// TIA Portal project "3_Queue_of_Items" (V19)

(* hardware
DEVICE "S7-1500/ET200MP station_1"  S7-1500 station
   slot 0: "Rail_0"  Rack  6ES7 590-1***0-0AA0
   slot 1: "PLC_1"  CPU 1513-1 PN  6ES7 513-1AL02-0AB0  V2.9
      slot 3: "CPU display_1"  6ES7591-1AA00-0AA0
      slot 32768: "PROFINET interface_1"  X1
         slot 32769: "Port_1"  X1 P1
         slot 32770: "Port_2"  X1 P2
      slot 34817: "Virtual CP interface port_1"  Virtual CP interface port  Virtual CP interface port
*)

// ===== PLC "PLC_1"  CPU 1513-1 PN =====

VAR_GLOBAL   // PLC tag table "Default tag table"
   "NGE_I0.3_Buffer" AT %M0.0 : Bool;
   "PE_Buffer_Conveyor" AT %M0.1 : Bool;
   "NE_Buffer_Conveyor" AT %M0.2 : Bool;
   "NE_Entry" AT %M0.3 : Bool;
   "NE_Exit" AT %M0.4 : Bool;
END_VAR

VAR_GLOBAL   // PLC tag table "Tag table from XML_1"
   "Start Button 1" AT %I0.0 : Bool;
   "Stop Button 1" AT %I0.1 : Bool;
   "Item Ready" AT %I0.2 : Bool;
   "At Entry" AT %I0.3 : Bool;
   "At Exit" AT %I0.4 : Bool;
   "Start Button 1 (Light)" AT %Q0.0 : Bool;
   "Stop Button 1 (Light)" AT %Q0.1 : Bool;
   "Entry conveyor" AT %Q0.2 : Bool;
   "Buffer conveyor" AT %Q0.3 : Bool;
   "Digital Display 1" AT %QD30 : DInt;
END_VAR

// folder: System blocks/Program resources

DATA_BLOCK "IEC_Counter_0_DB"   // DB1
{ S7_Optimized_Access := 'TRUE' }
AUTHOR : Simatic
FAMILY : IEC
NAME : CNTR
VERSION : 1.0
// stored: InstanceOfName IEC_COUNTER
"IEC_COUNTER"
BEGIN
END_DATA_BLOCK

DATA_BLOCK "IEC_Counter_0_DB_1"   // DB2
{ S7_Optimized_Access := 'TRUE' }
AUTHOR : Simatic
FAMILY : IEC
NAME : CNTR
VERSION : 1.0
// stored: InstanceOfName IEC_COUNTER
"IEC_COUNTER"
BEGIN
END_DATA_BLOCK

// folder: (top level)

ORGANIZATION_BLOCK "Main"   // OB1, LAD, ProgramCycle
TITLE = "Main Program Sweep (Cycle)"
{ S7_Optimized_Access := 'TRUE' }
VERSION : 0.1
   VAR_INPUT
      Initial_Call : Bool;   // Initial call of this OB
      Remanence : Bool;   // =True, if remanent data are available
   END_VAR
   VAR_TEMP   // added for the SCL form of the ladder/FBD networks
      _w1 : Bool;
      _w2 : Bool;
   END_VAR
BEGIN

REGION Network 1: Initial condition
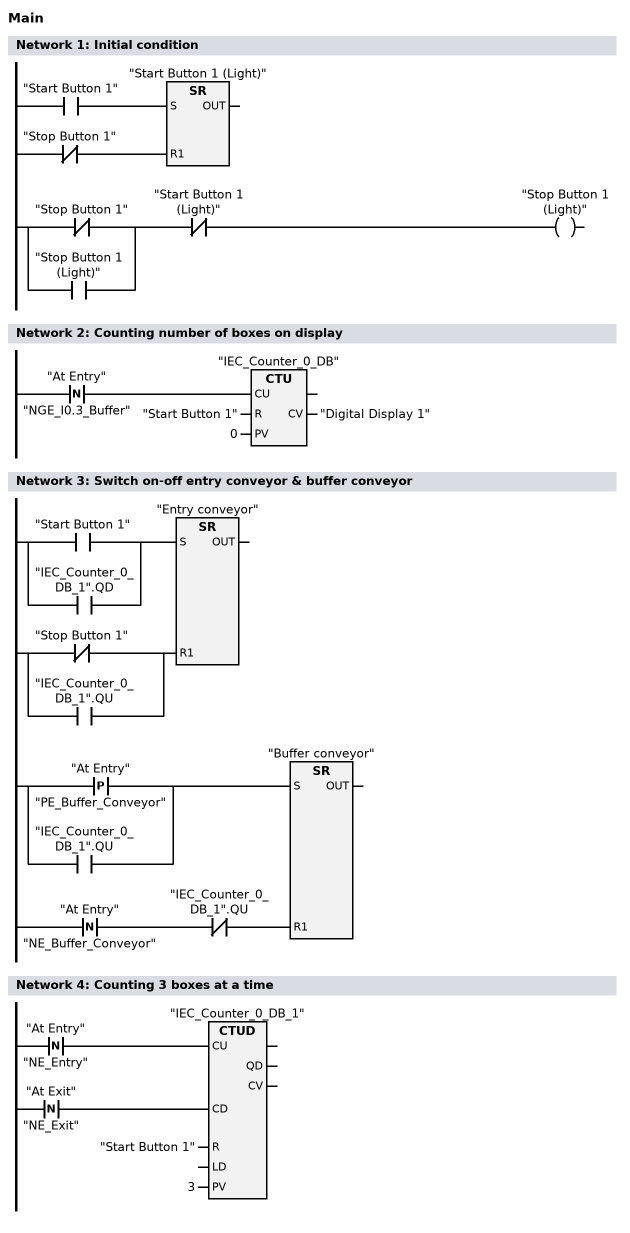
   RUNG wire#powerrail
      Contact( "Start Button 1" )
      S_SR(operand := "Start Button 1 (Light)", r1 := wire#w1)
   END_RUNG
   RUNG wire#powerrail
      I_Contact( "Stop Button 1" )
   END_RUNG wire#w1
   RUNG wire#powerrail
      I_Contact( "Stop Button 1" )
      wire#w2
      I_Contact( "Start Button 1 (Light)" )
      Coil( "Stop Button 1 (Light)" )
   END_RUNG
   RUNG wire#powerrail
      Contact( "Stop Button 1 (Light)" )
   END_RUNG wire#w2
   // the same network as SCL:
   IF "Start Button 1" THEN
       "Start Button 1 (Light)" := TRUE;   // SR flip-flop
   END_IF;
   IF NOT "Stop Button 1" THEN "Start Button 1 (Light)" := FALSE; END_IF;
   "Stop Button 1 (Light)" := (NOT "Stop Button 1" OR "Stop Button 1 (Light)") AND NOT "Start Button 1 (Light)";
END_REGION

REGION Network 2: Counting number of boxes on display
   #_w1 := NOT "At Entry" AND "NGE_I0.3_Buffer";   // falling edge of "At Entry"
   "NGE_I0.3_Buffer" := "At Entry";
   "IEC_Counter_0_DB".CTU(CU := #_w1, R := "Start Button 1", PV := 0, CV => "Digital Display 1");
END_REGION

REGION Network 3: Switch on-off entry conveyor & buffer conveyor
   RUNG wire#powerrail
      Contact( "Start Button 1" )
      wire#w1
      S_SR(operand := "Entry conveyor", r1 := wire#w2)
   END_RUNG
   RUNG wire#powerrail
      Contact( "IEC_Counter_0_DB_1".QD )
   END_RUNG wire#w1
   RUNG wire#powerrail
      I_Contact( "Stop Button 1" )
   END_RUNG wire#w2
   RUNG wire#powerrail
      Contact( "IEC_Counter_0_DB_1".QU )
   END_RUNG wire#w2
   RUNG wire#powerrail
      P_Contact(operand := "At Entry", bit := "PE_Buffer_Conveyor")
      wire#w3
      S_SR(operand := "Buffer conveyor", r1 := wire#w4)
   END_RUNG
   RUNG wire#powerrail
      Contact( "IEC_Counter_0_DB_1".QU )
   END_RUNG wire#w3
   RUNG wire#powerrail
      N_Contact(operand := "At Entry", bit := "NE_Buffer_Conveyor")
      I_Contact( "IEC_Counter_0_DB_1".QU )
   END_RUNG wire#w4
   // the same network as SCL:
   IF "Start Button 1" OR "IEC_Counter_0_DB_1".QD THEN
       "Entry conveyor" := TRUE;   // SR flip-flop
   END_IF;
   IF NOT "Stop Button 1" OR "IEC_Counter_0_DB_1".QU THEN "Entry conveyor" := FALSE; END_IF;
   #_w1 := "At Entry" AND NOT "PE_Buffer_Conveyor";   // rising edge of "At Entry"
   "PE_Buffer_Conveyor" := "At Entry";
   #_w2 := NOT "At Entry" AND "NE_Buffer_Conveyor";   // falling edge of "At Entry"
   "NE_Buffer_Conveyor" := "At Entry";
   IF #_w1 OR "IEC_Counter_0_DB_1".QU THEN
       "Buffer conveyor" := TRUE;   // SR flip-flop
   END_IF;
   IF #_w2 AND NOT "IEC_Counter_0_DB_1".QU THEN "Buffer conveyor" := FALSE; END_IF;
END_REGION

REGION Network 4: Counting 3 boxes at a time
   #_w1 := NOT "At Entry" AND "NE_Entry";   // falling edge of "At Entry"
   "NE_Entry" := "At Entry";
   #_w2 := NOT "At Exit" AND "NE_Exit";   // falling edge of "At Exit"
   "NE_Exit" := "At Exit";
   "IEC_Counter_0_DB_1".CTUD(CU := #_w1, CD := #_w2, R := "Start Button 1", PV := 3);
END_REGION
END_ORGANIZATION_BLOCK